(* LS Electric XG5000 project: PID *)
(* PLC LSPLC *)

PROGRAM NewProgram (* task: 스캔 프로그램 *)
VAR
    AP재시작 : BOOL;
    AT목표값 : INT;
    AT시작 : BOOL;
    DA출력데이터 : INT;
    INST : PIDRUN;
    mm : BOOL;
    PID목표값 : INT;
    PID운전시작 : BOOL;
    목표값 : BOOL;
    외부PV : BOOL;
    외부온도값 : INT;
END_VAR
VAR
    _e1 : R_TRIG;
    _e2 : R_TRIG;
END_VAR

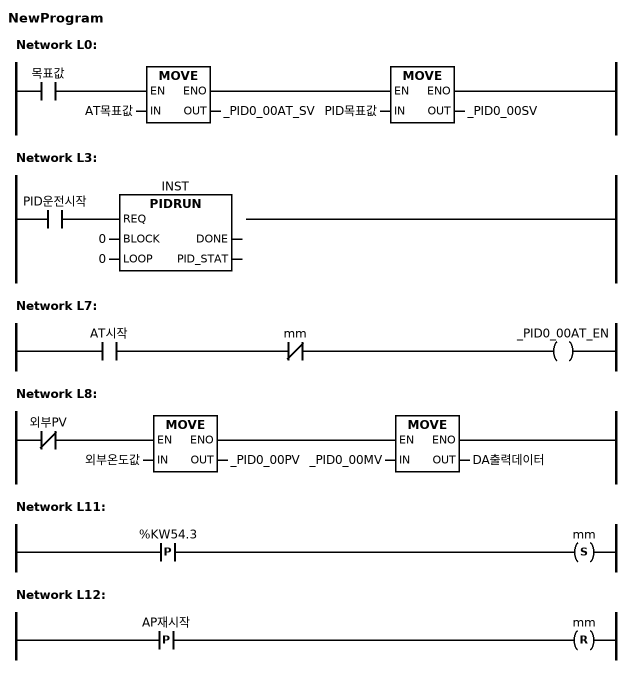
(* Rung L0 *)
IF 목표값 THEN
    _PID0_00AT_SV := AT목표값;
    _PID0_00SV := PID목표값;
END_IF;
(* Rung L3 *)
INST(REQ := PID운전시작, BLOCK := 0, LOOP := 0);
(* Rung L7 *)
_PID0_00AT_EN := AT시작 AND NOT mm;
(* Rung L8 *)
IF NOT 외부PV THEN
    _PID0_00PV := 외부온도값;
    DA출력데이터 := _PID0_00MV;
END_IF;
(* Rung L11 *)
_e1(CLK := %KW54.3);
IF _e1.Q THEN mm := TRUE; END_IF;
(* Rung L12 *)
_e2(CLK := AP재시작);
IF _e2.Q THEN mm := FALSE; END_IF;
END_PROGRAM